FUNCTION_BLOCK int_arr_to_real_1
VAR_INPUT
	array_pos_0 : WORD;
	array_pos_1 : WORD;
END_VAR
VAR_OUTPUT
	output : REAL;
END_VAR
VAR
	msb_hex: STRING(255);
	lsb_hex: STRING(255);
	concat_hex: STRING(255);
	cbData: UDINT;
	hex_byte_data:  ARRAY[0..3] OF BYTE;;
	uConvert : U_Convert;
END_VAR

msb_hex := WORD_TO_HEXSTR(in := array_pos_0, iPrecision := 4, bLoCase := FALSE);
lsb_hex := WORD_TO_HEXSTR(in := array_pos_1, iPrecision := 4, bLoCase := FALSE);	

concat_hex := CONCAT(STR1 := msb_hex , STR2 := lsb_hex );

cbData := HEXSTR_TO_DATA( concat_hex, ADR( hex_byte_data), SIZEOF( hex_byte_data ) );
			
uconvert.arrUDP_Data[3] := hex_byte_data[0];
uconvert.arrUDP_Data[2] := hex_byte_data[1];
uconvert.arrUDP_Data[1] := hex_byte_data[2];
uconvert.arrUDP_Data[0] := hex_byte_data[3];

output := uconvert.rReal;

END_FUNCTION_BLOCK

(* stored: Version 1.1.0.1, ProductVersion 3.1.4024.15
   POU int_arr_to_real_1: Id {986e71d7-8220-4703-b116-99ebe5f47bb9}, SpecialFunc None *)
